// TIA Portal V16 export
// export: Created 2021-11-12T13:33:15.2754748Z, ExportSetting WithDefaults, DisplayName Totally Integrated Automation Portal, DisplayVersion V16 Update 3, DisplayName TIA Portal Version Control Interface, DisplayVersion V16 Update 2, DisplayName TIA Portal Openness, DisplayVersion V16 Update 3, DisplayName SINAMICS Startdrive Advanced, DisplayVersion V16 Update 5, DisplayName SINAMICS Startdrive G130, G150, S120, S150, SINAMICS MV, S210, DisplayVersion V16 Update 5, DisplayName SINAMICS Startdrive G110M, G120, G120C, G120D, G120P, G115D, DisplayVersion V16 Update 5, DisplayName STEP 7 Professional, DisplayVersion V16 Update 3, DisplayName STEP 7 Safety, DisplayVersion V16, DisplayName WinCC UA Professional, DisplayVersion V16 Update 3
DATA_BLOCK "HMI_PARAM_Zone400"   // DB119
{ S7_Optimized_Access := 'TRUE'; DB_Accessible_From_OPC_UA := 'FALSE' }
VERSION : 0.1
// stored: AutoNumber true, DBAccessibleFromOPCUA false, IsOnlyStoredInLoadMemory false, IsRetainMemResEnabled false, IsWriteProtectedInAS false, MemoryReserve 100
   VAR
      Mode : "UDT_Zone_Parameter";   // Parameters of zone 400
      Station410_Mode : "UDT_Station_Parameter";   // Parameters of station 410
      Station420_Mode : "UDT_Station_Parameter";   // Parameters of station 420
      Station430_Mode : "UDT_Station_Parameter";   // Parameters of station 430
      Station440_Mode : "UDT_Station_Parameter";   // Parameters of station 440
      Station450_Mode : "UDT_Station_Parameter";   // Parameters of station 450
      Station460_Mode { S7_SetPoint := 'True'} : "UDT_Station_Parameter";   // Parameters of station 460
      StationTHM1_Mode { S7_SetPoint := 'True'} : "UDT_Station_Parameter";   // Parameters of station THM1
      StationTHM2_Mode { S7_SetPoint := 'True'} : "UDT_Station_Parameter";   // Parameters of station THM2
   END_VAR
BEGIN
   Mode.HMI1.FuncBtnPanelNr := 10;
   Mode.HMI2.FuncBtnPanelNr := 20;
   Mode.HMI3.FuncBtnPanelNr := 30;
END_DATA_BLOCK
